FUNCTION_BLOCK KMEANS
  {SET_ATTRIBUTE(OpcUa, SERVICE)}
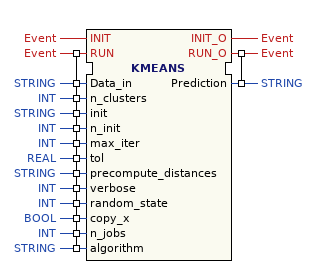
  EVENT_INPUT
    INIT;
    RUN WITH Data_in, n_clusters, init, n_init, max_iter, tol, precompute_distances, verbose, random_state, copy_x, n_jobs, algorithm; {SET_ATTRIBUTE(OpcUa, Method)}
  END_EVENT
  EVENT_OUTPUT
    INIT_O;
    RUN_O WITH Prediction;
  END_EVENT
  VAR_INPUT
    Data_in : STRING; {SET_ATTRIBUTE(OpcUa, Variable.RUN)}
    n_clusters : INT; {SET_ATTRIBUTE(OpcUa, Variable.RUN)}
    init : STRING; {SET_ATTRIBUTE(OpcUa, Variable.RUN)}
    n_init : INT; {SET_ATTRIBUTE(OpcUa, Variable.RUN)}
    max_iter : INT; {SET_ATTRIBUTE(OpcUa, Variable.RUN)}
    tol : REAL; {SET_ATTRIBUTE(OpcUa, Variable.RUN)}
    precompute_distances : STRING; {SET_ATTRIBUTE(OpcUa, Variable.RUN)}
    verbose : INT; {SET_ATTRIBUTE(OpcUa, Variable.RUN)}
    random_state : INT; {SET_ATTRIBUTE(OpcUa, Variable.RUN)}
    copy_x : BOOL; {SET_ATTRIBUTE(OpcUa, Variable.RUN)}
    n_jobs : INT; {SET_ATTRIBUTE(OpcUa, Variable.RUN)}
    algorithm : STRING; {SET_ATTRIBUTE(OpcUa, Variable.RUN)}
  END_VAR
  VAR_OUTPUT
    Prediction : STRING; {SET_ATTRIBUTE(OpcUa, Variable.RUN)}
  END_VAR
END_FUNCTION_BLOCK
